FUNCTION_BLOCK DeleteMe
VAR_INPUT
END_VAR
VAR_OUTPUT
END_VAR
VAR

END_VAR


(*  *********************************************************** *)
(*  LAP 2010/1 Kompressoranlage                                 *)
(*  *********************************************************** *)

DA.P1 := DI.S1;

END_FUNCTION_BLOCK

(* stored: Version 1.1.0.1, ProductVersion 3.1.4024.5
   POU DeleteMe: Id {f156885e-d892-4706-970d-8d2a74171c01}, SpecialFunc None *)
